// TIA Portal V16 export
// export: Created 2021-06-25T07:12:00.0552914Z, ExportSetting WithDefaults, DisplayName Totally Integrated Automation Portal, DisplayVersion V16, DisplayName TIA Portal Version Control Interface, DisplayVersion V16, DisplayName TIA Portal Openness, DisplayVersion V16, DisplayName STEP 7 Professional, DisplayVersion V16, DisplayName STEP 7 Safety, DisplayVersion V16, DisplayName WinCC Advanced, DisplayVersion V16
VAR_GLOBAL   // PLC tag table "Default tag table"
END_VAR
